// TIA Portal V20 export
TYPE "zu_CallData"
// stored: Access Published, Namespace CITI_Logic
   STRUCT
      Request : Bool;
      Acknowledge : Bool;
      Reset : Bool;
   END_STRUCT;
END_TYPE
